FUNCTION_BLOCK ENCODE_OPERATION_COMMAND (* Encodes an Operation Command word from RUN/DIRECTION, or a Fault Reset code on an explicit event *)
  (* Standard: 61499-1; Description: Copyright (c) 2026 HR Agrartechnik GmbH This program and the accompanying materials are made available under the terms of the Eclipse Public License 2.0 which is available at https://www.eclipse.org/legal/epl-2.0/ SPDX-License-Identifier: EPL-2.0 Generic building block for any VFD/drive whose Operation Command word follows the common Run/Direction/Stop + explicit Fault-Reset-override pattern (Modbus, CANopen PZD1, Profibus PPO, etc.). Named 'Operation Command', not 'Control Word' - the latter is CANopen-specific terminology, whereas 'Operation Command' is the vendor-neutral term used by e.g. the DELIXI H300 manual. All command codes are supplied by the caller via Parameter, so the block itself carries no brand-specific knowledge - only the encoding shape. *)
  (* Version 2.0, 2026-08-26, Franz Höpfinger, HR Agrartechnik GmbH, renamed from ENCODE_CONTROLWORD / CW_* / CONTROL_WORD to ENCODE_OPERATION_COMMAND / OC_* / OPERATION_COMMAND - Control Word is CANopen terminology *)
  (* Version 1.0, 2026-08-26, Franz Höpfinger, HR Agrartechnik GmbH, generalized from H300_ENCODE_CONTROLWORD - initial API and implementation *)
  PACKAGE logiBUS::drives;
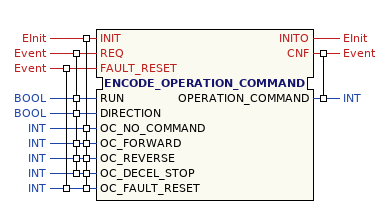
  EVENT_INPUT
    INIT : EInit WITH OC_NO_COMMAND, OC_FORWARD, OC_REVERSE, OC_DECEL_STOP, OC_FAULT_RESET; (* Init Request *)
    REQ WITH RUN, DIRECTION, OC_FORWARD, OC_REVERSE, OC_DECEL_STOP; (* RUN/DIRECTION evaluated *)
    FAULT_RESET WITH OC_FAULT_RESET; (* Request the Fault Reset command code *)
  END_EVENT
  EVENT_OUTPUT
    INITO : EInit; (* Init Confirmation *)
    CNF WITH OPERATION_COMMAND; (* Operation Command updated *)
  END_EVENT
  VAR_INPUT
    RUN : BOOL; (* Run command *)
    DIRECTION : BOOL; (* FALSE=Forward, TRUE=Reverse *)
    OC_NO_COMMAND : INT; (* Operation Command code for No Command / safe default (drive-specific, via Parameter) *)
    OC_FORWARD : INT; (* Operation Command code for Forward Run (drive-specific, via Parameter) *)
    OC_REVERSE : INT; (* Operation Command code for Reverse Run (drive-specific, via Parameter) *)
    OC_DECEL_STOP : INT; (* Operation Command code for Decelerated Stop (drive-specific, via Parameter) *)
    OC_FAULT_RESET : INT; (* Operation Command code for Fault Reset (drive-specific, via Parameter) *)
  END_VAR
  VAR_OUTPUT
    OPERATION_COMMAND : INT; (* Encoded Operation Command (target register content) *)
  END_VAR
  EC_STATES
    INIT : INIT -> INITO;
    REQ : REQ -> CNF;
    FAULT_RESET : FAULT_RESET -> CNF;
  END_STATES
  ALGORITHM INIT IN ST: (* Sets OPERATION_COMMAND to No Command before the first REQ/FAULT_RESET *)
OPERATION_COMMAND := OC_NO_COMMAND;
  END_ALGORITHM
  ALGORITHM REQ IN ST: (* Encodes RUN/DIRECTION as Forward/Reverse/Decelerated Stop command *)
IF RUN THEN
	IF DIRECTION THEN
		OPERATION_COMMAND := OC_REVERSE;
	ELSE
		OPERATION_COMMAND := OC_FORWARD;
	END_IF;
ELSE
	OPERATION_COMMAND := OC_DECEL_STOP;
END_IF;
  END_ALGORITHM
  ALGORITHM FAULT_RESET IN ST: (* Overwrites OPERATION_COMMAND once with the Fault Reset code, independent of RUN/DIRECTION *)
OPERATION_COMMAND := OC_FAULT_RESET;
  END_ALGORITHM
END_FUNCTION_BLOCK
